TYPE ST_GCSpinAxisMoveAbsService :
STRUCT
	Ctrl : ST_GCSpinAxisMoveAbsCtrl;
	Status : ST_GCSpinAxisMoveAbsStatus;
END_STRUCT
END_TYPE

(* stored: Version 1.1.0.1, ProductVersion 3.1.4026.18
   DUT ST_GCSpinAxisMoveAbsService: Id {5e24cf64-844d-4d0a-84fa-35d46a874805} *)
